// TIA Portal V18 export
// export: Created 2026-06-05T07:40:23.4725839Z, ExportSetting WithDefaults, DisplayName Totally Integrated Automation Portal, DisplayVersion V18, DisplayName TIA Portal Openness, DisplayVersion V18, DisplayName TIA Portal Version Control Interface, DisplayVersion V18, DisplayName STEP 7 Professional, DisplayVersion V18, DisplayName STEP 7 Safety, DisplayVersion V18, DisplayName WinCC Professional, DisplayVersion V18
ORGANIZATION_BLOCK "Cyclic interrupt"   // OB30, LAD, CyclicInterrupt
{ S7_Optimized_Access := 'TRUE' }
VERSION : 0.1
// stored: AutoNumber true, IsIECCheckEnabled false, SetENOAutomatically false
   VAR_INPUT
      Initial_Call : Bool;   // Initial call of this OB
      Event_Count : Int;   // Events discarded
   END_VAR
BEGIN

REGION Network 1
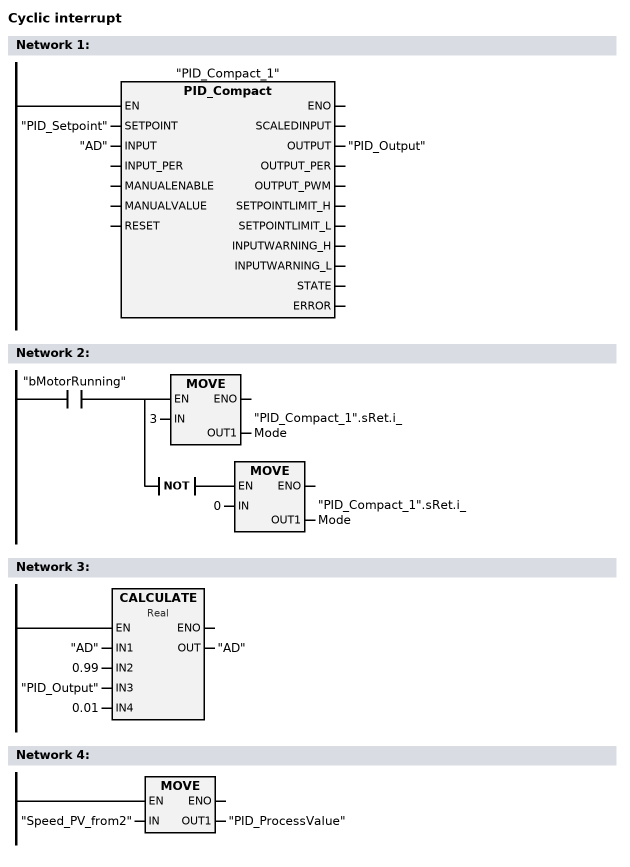
   RUNG wire#powerrail
      "PID_Compact_1".PID_Compact(Setpoint := "PID_Setpoint", Input := "AD", Input_PER :=, ManualEnable :=, ManualValue :=, Reset :=, ScaledInput =>, Output => "PID_Output", Output_PER =>, Output_PWM =>, SetpointLimit_H =>, SetpointLimit_L =>, InputWarning_H =>, InputWarning_L =>, State =>, Error =>)
   END_RUNG
   // the same network as SCL:
   "PID_Compact_1"(Setpoint := "PID_Setpoint", Input := "AD", Output => "PID_Output");   // PID_Compact
END_REGION

REGION Network 2
   RUNG wire#powerrail
      Contact( "bMotorRunning" )
      wire#w1
      Move(in := 3, out1 => "PID_Compact_1".sRet.i_Mode)
   END_RUNG
   RUNG wire#w1
      Not()
      Move(in := 0, out1 => "PID_Compact_1".sRet.i_Mode)
   END_RUNG
   // the same network as SCL:
   IF "bMotorRunning" THEN "PID_Compact_1".sRet.i_Mode := 3; END_IF;
   IF NOT "bMotorRunning" THEN "PID_Compact_1".sRet.i_Mode := 0; END_IF;
END_REGION

REGION Network 3
   RUNG wire#powerrail
      { S7_Templates := "SrcType := Real"; S7_Expression := "IN2*IN1 + IN4*IN3" } Calculate(in1 := "AD", in2 := 0.99, in3 := "PID_Output", in4 := 0.01, out => "AD")
   END_RUNG
   // the same network as SCL:
   "AD" := 0.99*"AD" + 0.01*"PID_Output";
END_REGION

REGION Network 4
   RUNG wire#powerrail
      Move(in := "Speed_PV_from2", out1 => "PID_ProcessValue")
   END_RUNG
   // the same network as SCL:
   "PID_ProcessValue" := "Speed_PV_from2";
END_REGION
END_ORGANIZATION_BLOCK
